TYPE ST_UserControl_Manual_Axis_Item_String :
STRUCT
	stName				: ST_Text;
	stPos				: ST_Text;
END_STRUCT
END_TYPE

(* stored: Version 1.1.0.1, ProductVersion 3.1.4024.11
   DUT ST_UserControl_Manual_Axis_Item_String: Id {576d2e21-d61c-4c44-8b13-ff6e73942069} *)
